FUNCTION_BLOCK PropotionalValve
VAR_INPUT
END_VAR
VAR_OUTPUT
END_VAR
VAR
	//Hardware
	AO_SetPressure AT %Q* : INT;
END_VAR

PROPERTY Pressure : INT
SET
AO_SetPressure := Pressure;
END_SET
END_PROPERTY

END_FUNCTION_BLOCK

(* stored: Version 1.1.0.1
   POU PropotionalValve: Id {e3b46589-8ac9-4c63-b0ed-f1d055628d04}, SpecialFunc None
   Property Pressure: Id {95fbf232-5040-4f3b-845c-3fbb4f1a834b}
   Set Set: Id {0bee4dec-8f9c-4294-a46e-80abd2176343} *)
